TYPE "UDT_MES_UnLoadData_ext"
VERSION : 0.1
   STRUCT
      "PLC.CheckSum" : Int;
      "PLC.PartTypeID" : Int;
      "PLC.PartTypeSN" : String[50];
      "PLC.SubPartSN" : String[50];
      "PLC.PartStatus" : DInt;
      "PLC.StatusBits2" : DInt;
      "PLC.Result" : Array[1..150] of Real;
      "MES.ErrorCode" : Int;
      "MES.ErrorMsg" : String[50];
   END_STRUCT;

END_TYPE

